// TIA Portal V18 export
FUNCTION_BLOCK "01_Speed_Control_SLS"   // FB7, F_LAD
{ S7_Optimized_Access := 'TRUE' }
   VAR_INPUT
      PH1 : Bool;   // Photoeye 1 input
      PH2 : Bool;   // Photoeye 2 input
      SORTER_RUNNING_MSC : Bool;   // Sorter running from MSC
      SLS_NOT_EN : Bool;   // SLS not enabled
      RESET { ExternalWritable := 'False'} : Bool;   // Reset alarms
      "MIN[time]" : Time;   // SLS Limit[ms] = Blade length[mm] / Speed[mm/s]
      "MAX[time]" : Time := T#4s;   // Sorter not moving
      "DelayRunning[time]" : Time := T#5s;   // Delay running status from sorter
   END_VAR
   VAR_OUTPUT
      SPEED_ZERO : Bool;   // Sorter stopped
      SPEED_TOOHIGH : Bool;   // Sorter speed too high ( not tested)
      "PH1 Broken" : Bool;   // Photoeye 1 broken
      "PH2 Broken" : Bool;   // Photoeye 2 broken
      ENC_BROKEN : Bool;   // Safety ancoder broken
   END_VAR
   VAR
      SR_RESET { ExternalWritable := 'False'} : Bool;
      Time_Limit : Time := T#10s;
      TON_SLS_T_PH1 : TON;
      TON_SLS_T_PH2 : TON;
      TOF_PH1_WORKING : TOF;
      TOF_PH2_WORKING : TOF;
      TON_SORTER_STOP : TON;
      TON_TIMEOUT_COUNT : TON;
      TON_DELAY_RUNNING_STATUS : TON;
      CTU_SLS_PH1 : CTU;
      CTU_SLS_PH2 : CTU;
      PH1_FE : Bool;
      PH1_RE : Bool;
      PH2_FE : Bool;
      PH2_RE : Bool;
      PH1_ET : Time;
      PH2_ET : Time;
      BROKEN_FE : Bool;
   END_VAR
   VAR_TEMP
      t_SpeedTH_PH1 : Bool;
      t_SpeedTH_PH2 : Bool;
      t_Speed0_PH1 : Bool;
      t_Speed0_PH2 : Bool;
      t_PH1_FE : Bool;
      t_PH2_FE : Bool;
      t_PH1_RE : Bool;
      t_PH2_RE : Bool;
      t_PH1_BRK : Bool;
      t_PH2_BRK : Bool;
      t_SorterRunning : Bool;
      t_ENC_BRK : Bool;
   END_VAR
   VAR CONSTANT
      NUM_STH : Int := 3;   // Number of blades with speed too high in TIMEOUT_CTU time
      TIMEOUT_CTU : Time := T#5s;   // Deltatime to count number of blades too fast
   END_VAR
   VAR_TEMP   // added for the SCL form of the ladder/FBD networks
      _w1 : Bool;
      _w2 : Bool;
   END_VAR
BEGIN

REGION Network 1: Falling Edges
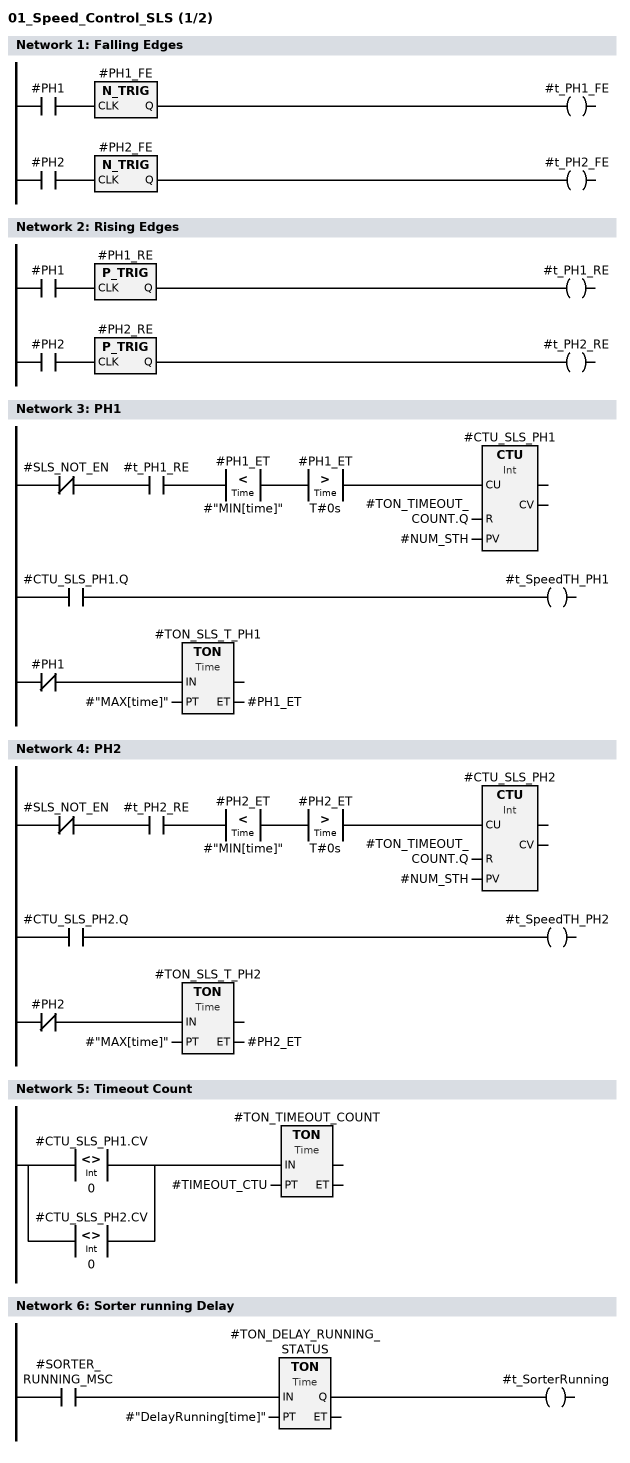
   RUNG wire#powerrail
      Contact( #PH1 )
      N_Trig( #PH1_FE )
      Coil( #t_PH1_FE )
   END_RUNG
   RUNG wire#powerrail
      Contact( #PH2 )
      N_Trig( #PH2_FE )
      Coil( #t_PH2_FE )
   END_RUNG
   // the same network as SCL:
   #_w1 := NOT #PH1 AND #PH1_FE;   // falling edge
   #PH1_FE := #PH1;
   #t_PH1_FE := #_w1;
   #_w2 := NOT #PH2 AND #PH2_FE;   // falling edge
   #PH2_FE := #PH2;
   #t_PH2_FE := #_w2;
END_REGION

REGION Network 2: Rising Edges
   RUNG wire#powerrail
      Contact( #PH1 )
      P_Trig( #PH1_RE )
      Coil( #t_PH1_RE )
   END_RUNG
   RUNG wire#powerrail
      Contact( #PH2 )
      P_Trig( #PH2_RE )
      Coil( #t_PH2_RE )
   END_RUNG
   // the same network as SCL:
   #_w1 := #PH1 AND NOT #PH1_RE;   // rising edge
   #PH1_RE := #PH1;
   #t_PH1_RE := #_w1;
   #_w2 := #PH2 AND NOT #PH2_RE;   // rising edge
   #PH2_RE := #PH2;
   #t_PH2_RE := #_w2;
END_REGION

REGION Network 3: PH1
   RUNG wire#powerrail
      I_Contact( #SLS_NOT_EN )
      Contact( #t_PH1_RE )
      { S7_Templates := "SrcType := Time" } LT_Contact(in1 := #PH1_ET, in2 := #"MIN[time]")
      { S7_Templates := "SrcType := Time" } GT_Contact(in1 := #PH1_ET, in2 := T#0s)
      { S7_Templates := "[value_type := Int, codedbool_type := DInt]" } #CTU_SLS_PH1.CTU(r := #TON_TIMEOUT_COUNT.Q, pv := #NUM_STH, cv =>)
   END_RUNG
   RUNG wire#powerrail
      Contact( #CTU_SLS_PH1.Q )
      Coil( #t_SpeedTH_PH1 )
   END_RUNG
   RUNG wire#powerrail
      I_Contact( #PH1 )
      { S7_Templates := "[time_type := Time, codedbool_type := DInt]" } #TON_SLS_T_PH1.TON(pt := #"MAX[time]", et => #PH1_ET)
   END_RUNG
   // the same network as SCL:
   #CTU_SLS_PH1.CTU(CU := NOT #SLS_NOT_EN AND #t_PH1_RE AND (#PH1_ET < #"MIN[time]") AND (#PH1_ET > T#0s),
                    R := #TON_TIMEOUT_COUNT.Q,
                    PV := #NUM_STH);
   #t_SpeedTH_PH1 := #CTU_SLS_PH1.Q;
   #TON_SLS_T_PH1.TON(IN := NOT #PH1, PT := #"MAX[time]", ET => #PH1_ET);
END_REGION

REGION Network 4: PH2
   RUNG wire#powerrail
      I_Contact( #SLS_NOT_EN )
      Contact( #t_PH2_RE )
      { S7_Templates := "SrcType := Time" } LT_Contact(in1 := #PH2_ET, in2 := #"MIN[time]")
      { S7_Templates := "SrcType := Time" } GT_Contact(in1 := #PH2_ET, in2 := T#0s)
      { S7_Templates := "[value_type := Int, codedbool_type := DInt]" } #CTU_SLS_PH2.CTU(r := #TON_TIMEOUT_COUNT.Q, pv := #NUM_STH, cv =>)
   END_RUNG
   RUNG wire#powerrail
      Contact( #CTU_SLS_PH2.Q )
      Coil( #t_SpeedTH_PH2 )
   END_RUNG
   RUNG wire#powerrail
      I_Contact( #PH2 )
      { S7_Templates := "[time_type := Time, codedbool_type := DInt]" } #TON_SLS_T_PH2.TON(pt := #"MAX[time]", et => #PH2_ET)
   END_RUNG
   // the same network as SCL:
   #CTU_SLS_PH2.CTU(CU := NOT #SLS_NOT_EN AND #t_PH2_RE AND (#PH2_ET < #"MIN[time]") AND (#PH2_ET > T#0s),
                    R := #TON_TIMEOUT_COUNT.Q,
                    PV := #NUM_STH);
   #t_SpeedTH_PH2 := #CTU_SLS_PH2.Q;
   #TON_SLS_T_PH2.TON(IN := NOT #PH2, PT := #"MAX[time]", ET => #PH2_ET);
END_REGION

REGION Network 5: Timeout Count
   RUNG wire#powerrail
      { S7_Templates := "SrcType := Int" } NE_Contact(in1 := #CTU_SLS_PH1.CV, in2 := 0)
      wire#w1
      { S7_Templates := "[time_type := Time, codedbool_type := DInt]" } #TON_TIMEOUT_COUNT.TON(pt := #TIMEOUT_CTU, et =>)
   END_RUNG
   RUNG wire#powerrail
      { S7_Templates := "SrcType := Int" } NE_Contact(in1 := #CTU_SLS_PH2.CV, in2 := 0)
   END_RUNG wire#w1
   // the same network as SCL:
   #TON_TIMEOUT_COUNT.TON(IN := (#CTU_SLS_PH1.CV <> 0) OR (#CTU_SLS_PH2.CV <> 0), PT := #TIMEOUT_CTU);
END_REGION

REGION Network 6: Sorter running Delay
   RUNG wire#powerrail
      Contact( #SORTER_RUNNING_MSC )
      { S7_Templates := "[time_type := Time, codedbool_type := DInt]" } #TON_DELAY_RUNNING_STATUS.TON(pt := #"DelayRunning[time]", et =>)
      Coil( #t_SorterRunning )
   END_RUNG
   // the same network as SCL:
   #TON_DELAY_RUNNING_STATUS.TON(IN := #SORTER_RUNNING_MSC, PT := #"DelayRunning[time]");
   #t_SorterRunning := #TON_DELAY_RUNNING_STATUS.Q;
END_REGION

REGION Network 7: Speed too high
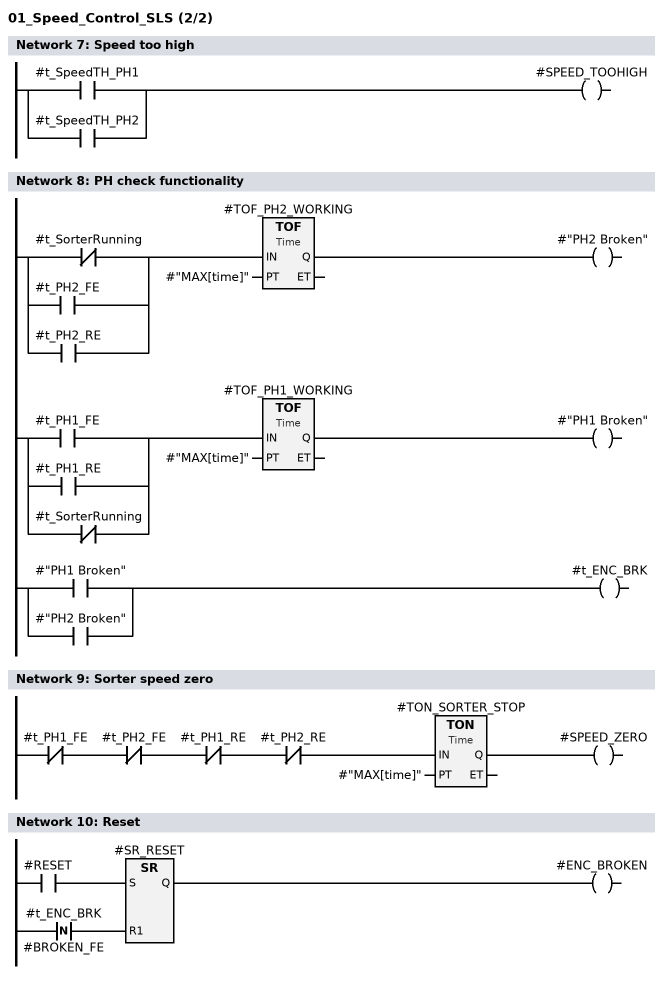
   RUNG wire#powerrail
      Contact( #t_SpeedTH_PH1 )
      wire#w1
      Coil( #SPEED_TOOHIGH )
   END_RUNG
   RUNG wire#powerrail
      Contact( #t_SpeedTH_PH2 )
   END_RUNG wire#w1
   // the same network as SCL:
   #SPEED_TOOHIGH := #t_SpeedTH_PH1 OR #t_SpeedTH_PH2;
END_REGION

REGION Network 8: PH check functionality
   RUNG wire#powerrail
      I_Contact( #t_SorterRunning )
      wire#w1
      { S7_Templates := "[time_type := Time, codedbool_type := DInt]" } #TOF_PH2_WORKING.TOF(pt := #"MAX[time]", et =>)
      Coil( #"PH2 Broken" )
   END_RUNG
   RUNG wire#powerrail
      Contact( #t_PH2_FE )
   END_RUNG wire#w1
   RUNG wire#powerrail
      Contact( #t_PH2_RE )
   END_RUNG wire#w1
   RUNG wire#powerrail
      Contact( #t_PH1_FE )
      wire#w2
      { S7_Templates := "[time_type := Time, codedbool_type := DInt]" } #TOF_PH1_WORKING.TOF(pt := #"MAX[time]", et =>)
      Coil( #"PH1 Broken" )
   END_RUNG
   RUNG wire#powerrail
      Contact( #t_PH1_RE )
   END_RUNG wire#w2
   RUNG wire#powerrail
      I_Contact( #t_SorterRunning )
   END_RUNG wire#w2
   RUNG wire#powerrail
      Contact( #"PH1 Broken" )
      wire#w3
      Coil( #t_ENC_BRK )
   END_RUNG
   RUNG wire#powerrail
      Contact( #"PH2 Broken" )
   END_RUNG wire#w3
   // the same network as SCL:
   #TOF_PH2_WORKING.TOF(IN := NOT #t_SorterRunning OR #t_PH2_FE OR #t_PH2_RE, PT := #"MAX[time]");
   #"PH2 Broken" := #TOF_PH2_WORKING.Q;
   #TOF_PH1_WORKING.TOF(IN := #t_PH1_FE OR #t_PH1_RE OR NOT #t_SorterRunning, PT := #"MAX[time]");
   #"PH1 Broken" := #TOF_PH1_WORKING.Q;
   #t_ENC_BRK := #"PH1 Broken" OR #"PH2 Broken";
END_REGION

REGION Network 9: Sorter speed zero
   RUNG wire#powerrail
      I_Contact( #t_PH1_FE )
      I_Contact( #t_PH2_FE )
      I_Contact( #t_PH1_RE )
      I_Contact( #t_PH2_RE )
      { S7_Templates := "[time_type := Time, codedbool_type := DInt]" } #TON_SORTER_STOP.TON(pt := #"MAX[time]", et =>)
      Coil( #SPEED_ZERO )
   END_RUNG
   // the same network as SCL:
   #TON_SORTER_STOP.TON(IN := NOT #t_PH1_FE AND NOT #t_PH2_FE AND NOT #t_PH1_RE AND NOT #t_PH2_RE,
                        PT := #"MAX[time]");
   #SPEED_ZERO := #TON_SORTER_STOP.Q;
END_REGION

REGION Network 10: Reset
   RUNG wire#powerrail
      Contact( #RESET )
      S_SR(operand := #SR_RESET, r1 := wire#w1)
      Coil( #ENC_BROKEN )
   END_RUNG
   RUNG wire#powerrail
      N_Contact(operand := #t_ENC_BRK, bit := #BROKEN_FE)
   END_RUNG wire#w1
   // the same network as SCL:
   #_w1 := NOT #t_ENC_BRK AND #BROKEN_FE;   // falling edge of #t_ENC_BRK
   #BROKEN_FE := #t_ENC_BRK;
   IF #RESET THEN
       #SR_RESET := TRUE;   // SR flip-flop
   END_IF;
   IF #_w1 THEN #SR_RESET := FALSE; END_IF;
   #ENC_BROKEN := #SR_RESET;
END_REGION
END_FUNCTION_BLOCK
